FUNCTION_BLOCK BfbIDMTCurve
  (* Standard: 61499-2 *)
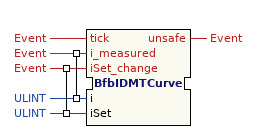
  EVENT_INPUT
    tick;
    i_measured WITH i;
    iSet_change WITH iSet;
  END_EVENT
  EVENT_OUTPUT
    unsafe;
  END_EVENT
  VAR_INPUT
    i : ULINT;
    iSet : ULINT;
  END_VAR
  VAR
    v : ULINT := 0;
    thresh : ULINT := 0;
    K : ULINT := 10000;
    B : ULINT := 135;
  END_VAR
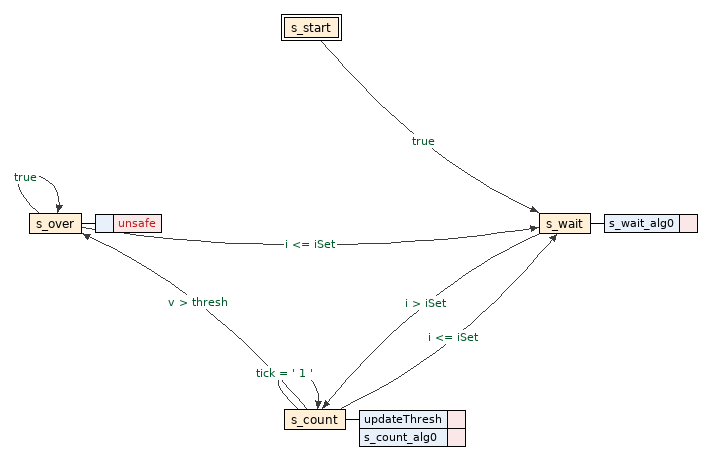
  EC_STATES
    s_start;
    s_wait : s_wait_alg0;
    s_count : updateThresh, s_count_alg0;
    s_over : -> unsafe;
  END_STATES
  EC_TRANSITIONS
    s_start TO s_wait := true;
    s_wait TO s_count := i > iSet;
    s_count TO s_wait := i <= iSet;
    s_count TO s_over := v > thresh;
    s_count TO s_count := tick = ' 1 ';
    s_over TO s_wait := i <= iSet;
    s_over TO s_over := true;
  END_TRANSITIONS
  ALGORITHM s_wait_alg0 IN VHDL:
v <= 0;
  END_ALGORITHM
  ALGORITHM s_count_alg0 IN VHDL:
v <= v + 1;
  END_ALGORITHM
  ALGORITHM updateThresh IN VHDL:
        thresh <= ((K*B) / ((I_mA / Iset_mA) - 1));
  END_ALGORITHM
END_FUNCTION_BLOCK
